FUNCTION derivcvar_M_p_t2: REAL
{ S7_Optimized_Access := 'false' }
    VAR_INPUT
        state: STATE;
    END_VAR

BEGIN
    derivcvar_M_p_t2 := 2.0;
END_FUNCTION
